{attribute 'qualified_only'}
VAR_GLOBAL
	
	myArray : ARRAY [0..10] OF MyStructure;
	
END_VAR

(* stored: Version 1.1.0.1, ProductVersion 3.1.4024.12
   GVL GVL: Id {e0d64cab-5156-4dc8-b883-b1bc41637862} *)
